// TIA Portal V18 export
// export: Created 2025-12-01T12:38:00.044048Z, ExportSetting None, DisplayName Totally Integrated Automation Portal, DisplayVersion V18 Update 5, DisplayName TIA Portal Openness, DisplayVersion V18 Update 5, DisplayName TIA Portal Teamcenter Gateway, DisplayVersion V18, DisplayName TIA Portal Version Control Interface, DisplayVersion V18, DisplayName STEP 7 Professional, DisplayVersion V18 Update 5, DisplayName STEP 7 Safety, DisplayVersion V18, DisplayName WinCC Professional, DisplayVersion V18 Update 5
DATA_BLOCK "DiagnosticDataBlock"   // DB3001
{ S7_Optimized_Access := 'FALSE' }
// stored: AutoNumber false
   VAR RETAIN
      DP : Struct
         DPReadStatus : Int;
         Status : Array[0..1023] of Bool;
      END_STRUCT;
      Profinet : Struct
         PNReadStatus : Int;
         Status : Array[0..1023] of Bool;
      END_STRUCT;
   END_VAR
BEGIN
   // DP.Status[0] : PLC-CPU
   // DP.Status[1] : Remote IO/ET200SP
   // DP.Status[2] : Festo Bus Coupler/总线耦合器
   // DP.Status[3] : CC-LINK
   // DP.Status[4] : Keyence Safety PLC
   // DP.Status[5] : Robot
   // DP.Status[6] : Keyence Laszer
   // DP.Status[7] : Balluff RFID
   // Profinet.Status[0] : ST70&ST80.PLC_CPU
   // Profinet.Status[1] : ST70&ST80.RFID
   // Profinet.Status[2] : ST70.Valves
   // Profinet.Status[3] : ST80.FCPN
   // Profinet.Status[4] : ST70.FCPN
   // Profinet.Status[5] : ST70.Screw
   // Profinet.Status[6] : CMMT-AS
   // Profinet.Status[7] : ST80.Screw
   // Profinet.Status[8] : ST80.Valves
END_DATA_BLOCK
